Universal Robots PolyScope program: xy.urp

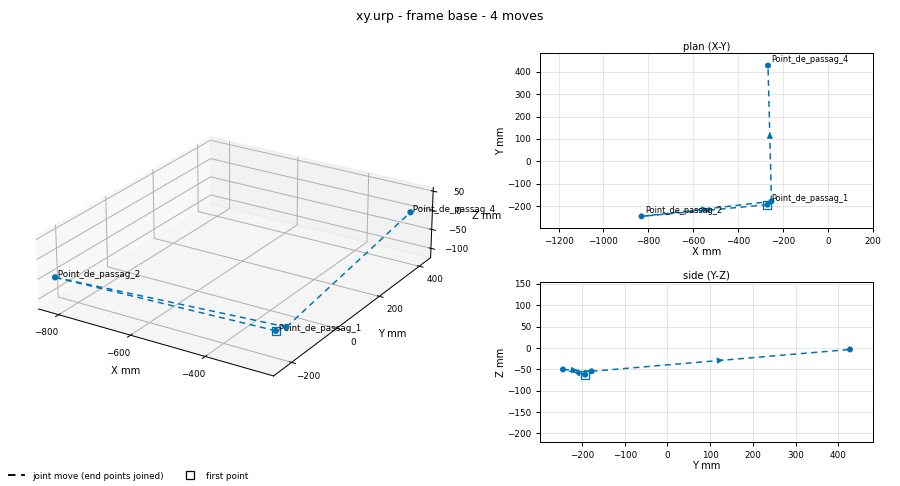
[picture p0: tool path of xy.urp in frame base, 4 of 4 moves have a stored position in this frame; points joined in program order, loops and branches not executed]
ProgramRoot directory=/programs; kinematics=(a=[0, -0.425, -0.39225, 0, 0, 0], d=[0.08916, 0, 0, 0.10915, 0.09465, 0.0823], alpha=[1.5708, 0, 0, 1.5708, -1.5708, 0], deltaTheta=[0, 0, 0, 0, 0, 0], status=notInitialized); name=xy; programVersion=(project__name=PolyScope, major__version=1, minor__version=6, svn__revision=9671, build__date=Dec 17 2012, 15:17:18); robotEnvironmentFileName=default
  MainProgram cartesianAcceleration=1.2; cartesianSpeed=0.25; jointAcceleration=1.3962634015954636; jointSpeed=1.0471975511965976; moveAsFastAsPossible=true; sharedProcessMoveBlendRadius=0.025; featureReference=(installationNameReference=Base); motionType=JOINT_SPACE
    Move cartesianAcceleration=1.2; cartesianSpeed=0.25; jointAcceleration=1.3962634015954636; jointSpeed=1.0471975511965976; moveAsFastAsPossible=true; sharedProcessMoveBlendRadius=0.025; featureReference=(installationNameReference=Base); motionType=JOINT_SPACE
      Waypoint blendRadius=0.05; cartesianAcceleration=1.2; cartesianSpeed=0.25; jointAcceleration=1.3962634015954636; jointSpeed=1.0471975511965976; nextMotionTime=2.0; stoppoint=true; useSharedBlendParameter=true; useSharedParameters=true; position=TCP in base x=-268.93 y=-192.842 z=-62.438 mm, rx=1.5707 ry=-0.028 rz=0.0329 rad; joints [0.296, -52.031, 140.263, -85.919, 0.117, -0.09] deg; positionType=FIXED_POSITION; waypointPoseInFeatureCoordinates=(pos=(x=-0.2689298869201141, y=-0.19284221705618498, z=-0.06243828013437344), rot=(x=1.5707231670046777, y=-0.028016119956013583, z=0.03292797839420235)); name=Point_de_passag_1
      Waypoint blendRadius=0.05; cartesianAcceleration=1.2; cartesianSpeed=0.25; jointAcceleration=1.3962634015954636; jointSpeed=1.0471975511965976; nextMotionTime=2.0; stoppoint=true; useSharedBlendParameter=true; useSharedParameters=true; position=TCP in base x=-830.216 y=-244.809 z=-50.109 mm, rx=1.5573 ry=0.1938 rz=-0.1003 rad; joints [3.651, -8.369, 26.354, -50.055, 0.251, 21.322] deg; positionType=FIXED_POSITION; waypointPoseInFeatureCoordinates=(pos=(x=-0.8302155911373357, y=-0.24480883237052598, z=-0.050109217612791954), rot=(x=1.5573297191328386, y=0.19377863283917607, z=-0.10028260619478566)); name=Point_de_passag_2
      Waypoint blendRadius=0.05; cartesianAcceleration=1.2; cartesianSpeed=0.25; jointAcceleration=1.3962634015954636; jointSpeed=1.0471975511965976; nextMotionTime=2.0; stoppoint=true; useSharedBlendParameter=true; useSharedParameters=true; position=TCP in base x=-250.91 y=-178.023 z=-54.508 mm, rx=1.5128 ry=0.0905 rz=0.0393 rad; joints [-2.92, -51.138, 137.929, -64.414, -8.369, -24.179] deg; positionType=FIXED_POSITION; waypointPoseInFeatureCoordinates=(pos=(x=-0.2509100728206708, y=-0.17802341234147542, z=-0.054507755332040136), rot=(x=1.5127817176820126, y=0.09046542131786774, z=0.03926926592948711)); name=Point_de_passag_3
      Waypoint blendRadius=0.05; cartesianAcceleration=1.2; cartesianSpeed=0.25; jointAcceleration=1.3962634015954636; jointSpeed=1.0471975511965976; nextMotionTime=2.0; stoppoint=true; useSharedBlendParameter=true; useSharedParameters=true; position=TCP in base x=-266.433 y=427.503 z=-3.331 mm, rx=1.5728 ry=0.0172 rz=0.1446 rad; joints [-72.514, -43.825, 91.959, -48.15, -78.419, 4.651] deg; positionType=FIXED_POSITION; waypointPoseInFeatureCoordinates=(pos=(x=-0.2664329605202211, y=0.42750343433070964, z=-0.003330890337358189), rot=(x=1.5727918829786869, y=0.017242543988799385, z=0.14459826032975268)); name=Point_de_passag_4
